// TIA Portal V20 export
// export: Created 2026-04-28T10:07:59.3999088Z, ExportSetting WithDefaults, DisplayName Totally Integrated Automation Portal, DisplayVersion V20, DisplayName TIA Portal Openness, DisplayVersion V20, DisplayName TIA Portal Version Control Interface, DisplayVersion V20, DisplayName SINAMICS Startdrive Advanced, DisplayVersion V20, DisplayName SINAMICS Startdrive G130, G150, S120, S150, SINAMICS MV, G220, S200, S210, DisplayVersion V20, DisplayName SINAMICS Startdrive G110M, G120, G120C, G120D, G120P, G115D, DisplayVersion V20, DisplayName STEP 7 Professional, DisplayVersion V20, DisplayName STEP 7 Safety, DisplayVersion V20, DisplayName WinCC Basic/Comfort/Advanced, DisplayVersion V20, DisplayName WinCC Unified, DisplayVersion V20
TYPE "PressenparameterVisu"
// stored: IsFailsafeCompliant false
   STRUCT
      xVersion01 : Bool;
      xZweiRegelkreise : Bool;
      xPH450_Hybrid : Bool;
      xDruckUerbers_Schl : Bool;
      xDue_Schliess_Visu : Bool;
      xContrPY1_1 : Bool;
      cPH450_RUP_PMR : Int;
      xOptSchwPlatte : Bool;
      xHY4_3neg : Bool;
      xTasterExtern : Bool;
      xOptMemP1_5 : Bool;
      xOberstempel_PR3_RK3 : Bool;
      xPoly_PIAB : Bool;
      tPoly_ON : Time;
      tPoly_Wait : Time;
      tPresseOeffnen_Verz : Time;
      t_Schaltp_P8_VerzT4_8 : Time;
      xIPEC : Bool;
      xMitRoboter : Bool;
      xOhneTransportBand : Bool;
      xMitVakuumPumpe : Bool;
      xIso_Limit_Ini : Bool;
      xMitExtPutz : Bool;
      xArtikelZaehlerTransport : Bool;
      xTrBand_Pr2_Option : Bool;
      xAbziehvorrOption : Bool;
      iVentilUeberw : Int;
      xPosition_US_Option : Bool;
      xTr2_Lang_Option : Bool;
      xExt_Entstaubung_Option : Bool;
      xOptionPB_Komm : Bool;
      xAbziehvorr_II_Option : Bool;
      xVorzentr_Seitlich_Option : Bool;
      acPosiFenster : Real;
      acAux05_Fuell : Real;
      uiRangeEilDrV : UInt;
      uiRangeEilDrR : UInt;
      uiRangeSysDr : UInt;
      uiRangeSchlDr : UInt;
      uiRangeIsostDr : UInt;
      uiRangePumpenD : UInt;
      uiRangeRSchlDr : UInt;
      acSchlZeit_T2_2 : String;
      acIsoStEin_T2_3 : Real;
      acStartb_Tx_0 : String;
      acVerzZentrFrei : String;
      acPosiIsoDr : String;
      ClosingPress : Array[1..15] of UInt;
      SR_RegP_Aufbau : Real;
      SR_RegI_Aufbau : Real;
      SR_RegD_Aufbau : Real;
      SR_RegP_Abbau : Real;
      SR_RegI_Abbau : Real;
      SR_RegD_Abbau : Real;
      SR_RegP_Aufbau_RK2 : Real;
      SR_RegI_Aufbau_RK2 : Real;
      SR_RegD_Aufbau_RK2 : Real;
      SR_RegP_Abbau_RK2 : Real;
      SR_RegI_Abbau_RK2 : Real;
      SR_RegD_Abbau_RK2 : Real;
      SR_P_SMC : Real;
      SR_I_SMC : Real;
      SR_D_SMC : Real;
      SR_AccUp_SMC : Real;
      SR_AccDwnSMC : Real;
   END_STRUCT;
END_TYPE
